// TIA Portal V20 export
TYPE "typeEMIdentMv"
// stored: Access Published
   STRUCT
      identMvEM : Array[0.."NO_OF_EM"] of "typeIdentMvHmi";
   END_STRUCT;
END_TYPE
